FUNCTION_BLOCK FB_System_FBT_425
VAR_INPUT
	Betrieb_Anford_auto		: BOOL;
	Regelung_Modus_auto		: USINT;
	Regelung_Sollw_auto		: REAL;
	Temp_Aussen				: REAL;
	Temp_Innen				: REAL;
END_VAR
VAR_OUTPUT
	{attribute 'OPC.UA.DA' := '1'}Steuerung				: ST_System_FBT_Steuerung;		
	{attribute 'OPC.UA.DA' := '1'}Stellwert				: ST_System_FBT_Stellwert;		
	{attribute 'OPC.UA.DA' := '1'}Zustand					: ST_System_FBT_Zustand;	
	{attribute 'OPC.UA.DA' := '1'}Parameter				: ST_System_FBT_Parameter;		
END_VAR
VAR
	Pumpe_425				: FB_PU;
	Stellventil_423			: FB_SVs;
	Stellventil_424			: FB_SVs;
	Regelventil_425			: FB_RV;

	Zustandscheck			: FB_System_FBT_Zustandscheck;
	Logik					: FB_System_FBT_Logik;
	Ablaufsteuerung			: FB_System_FBT_Ablaufsteuerung;
	Sollwertscheck			: FB_System_FBT_Sollwertscheck;
	Regelung				: FB_System_FBT_Regelung;
	Stellwertscheck			: FB_System_FBT_Stellwertscheck;

END_VAR
VAR // added by the converter: edge detectors and wires of the graphical bodies
    _w1, _w2 : ANY;
END_VAR

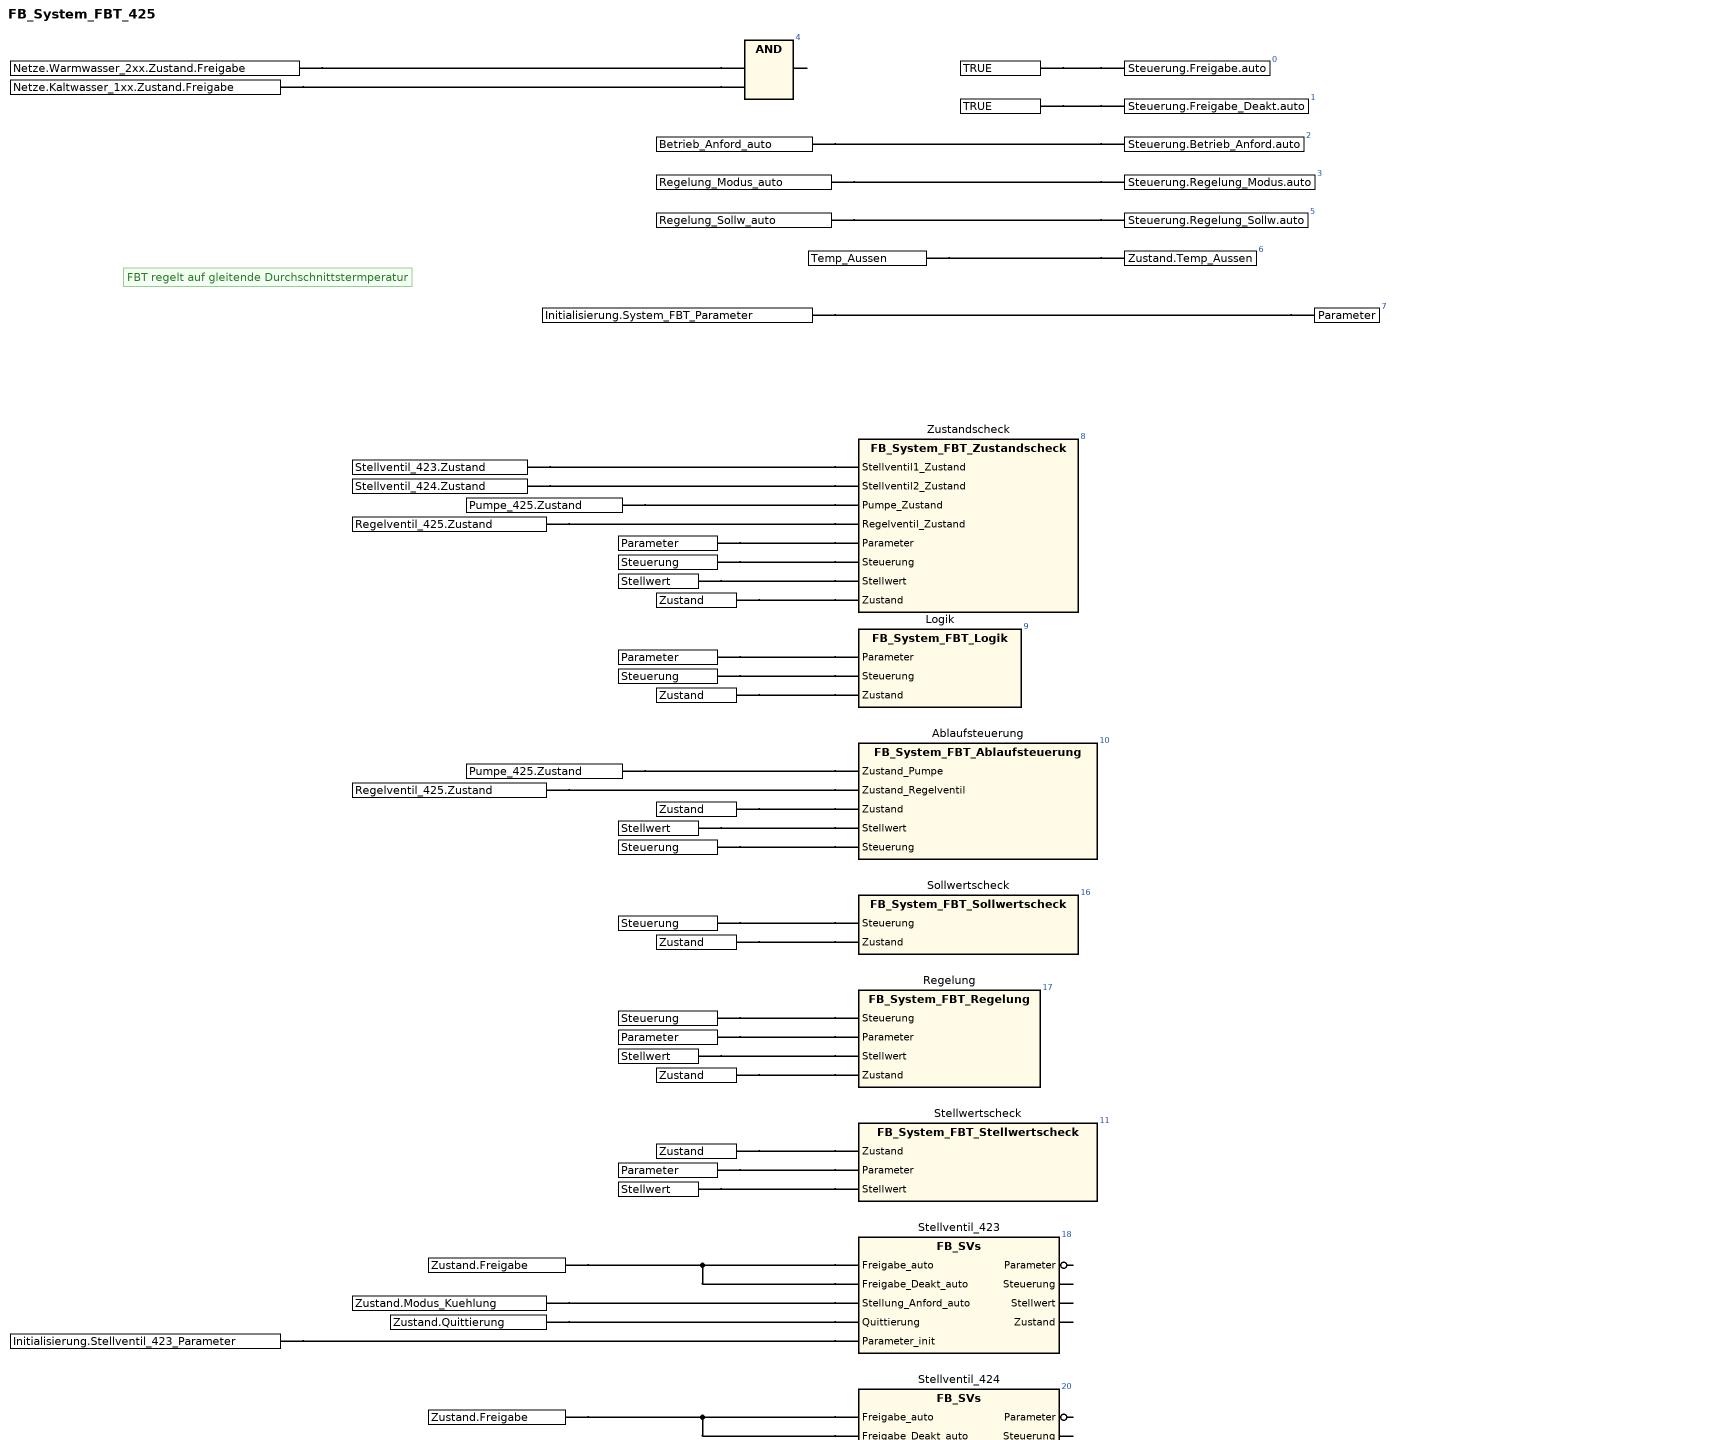
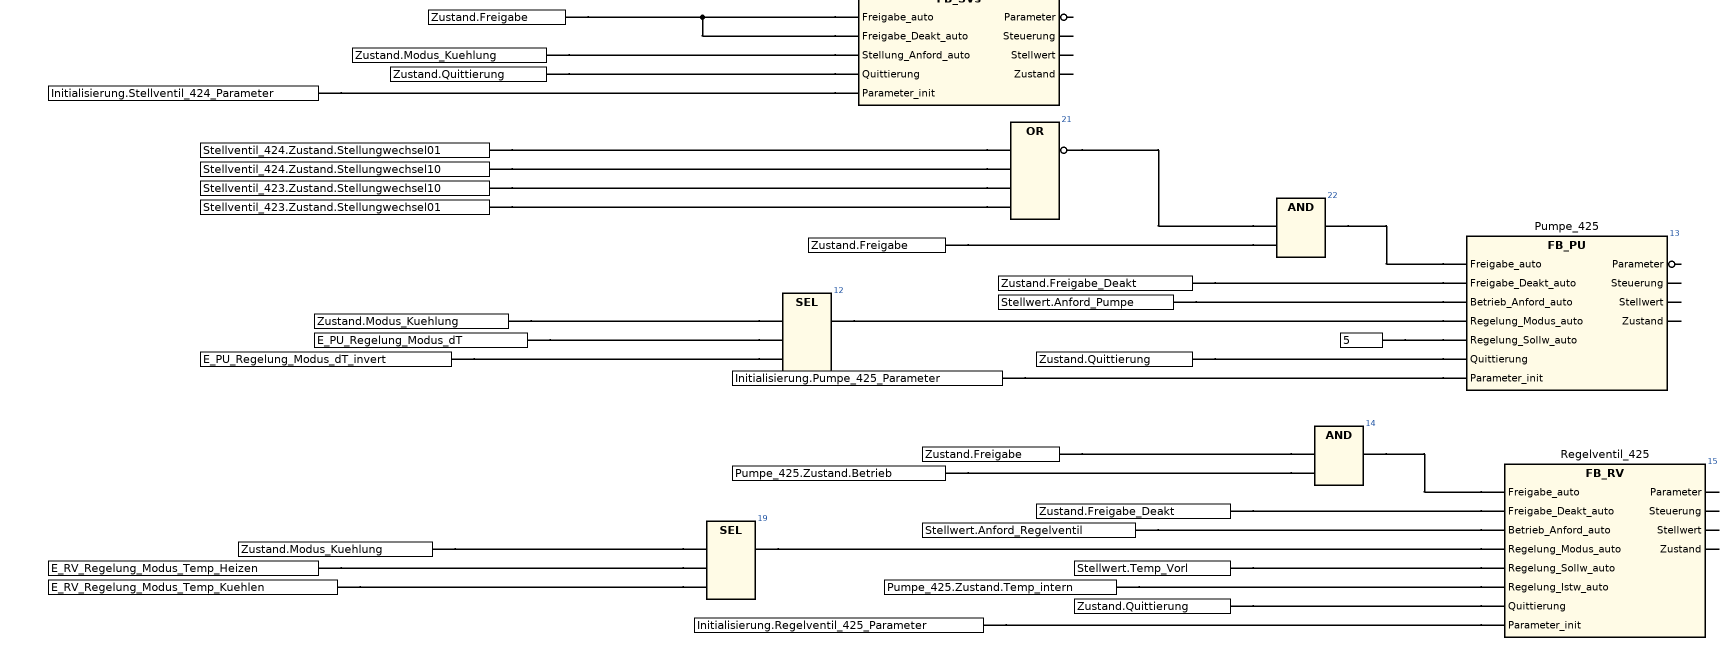
Steuerung.Freigabe.auto := TRUE;
Steuerung.Freigabe_Deakt.auto := TRUE;
Steuerung.Betrieb_Anford.auto := Betrieb_Anford_auto;
Steuerung.Regelung_Modus.auto := Regelung_Modus_auto;
(* Netze.Warmwasser_2xx.Zustand.Freigabe AND Netze.Kaltwasser_1xx.Zustand.Freigabe; result not used *)
Steuerung.Regelung_Sollw.auto := Regelung_Sollw_auto;
Zustand.Temp_Aussen := Temp_Aussen;
Parameter := Initialisierung.System_FBT_Parameter;
// FBT regelt auf gleitende Durchschnittstermperatur
Zustandscheck(
    Stellventil1_Zustand := Stellventil_423.Zustand,
    Stellventil2_Zustand := Stellventil_424.Zustand,
    Pumpe_Zustand := Pumpe_425.Zustand,
    Regelventil_Zustand := Regelventil_425.Zustand,
    Parameter := Parameter,
    Steuerung := Steuerung,
    Stellwert := Stellwert,
    Zustand := Zustand); // FB_System_FBT_Zustandscheck
Logik(Parameter := Parameter, Steuerung := Steuerung, Zustand := Zustand); // FB_System_FBT_Logik
Ablaufsteuerung(
    Zustand_Pumpe := Pumpe_425.Zustand,
    Zustand_Regelventil := Regelventil_425.Zustand,
    Zustand := Zustand,
    Stellwert := Stellwert,
    Steuerung := Steuerung); // FB_System_FBT_Ablaufsteuerung
Stellwertscheck(Zustand := Zustand, Parameter := Parameter, Stellwert := Stellwert); // FB_System_FBT_Stellwertscheck
Pumpe_425(
    Freigabe_auto := _w1,
    Freigabe_Deakt_auto := Zustand.Freigabe_Deakt,
    Betrieb_Anford_auto := Stellwert.Anford_Pumpe,
    Regelung_Modus_auto := SEL(Zustand.Modus_Kuehlung, E_PU_Regelung_Modus_dT, E_PU_Regelung_Modus_dT_invert),
    Regelung_Sollw_auto := 5,
    Quittierung := Zustand.Quittierung,
    Parameter_init := Initialisierung.Pumpe_425_Parameter); // FB_PU
Regelventil_425(
    Freigabe_auto := Zustand.Freigabe AND Pumpe_425.Zustand.Betrieb,
    Freigabe_Deakt_auto := Zustand.Freigabe_Deakt,
    Betrieb_Anford_auto := Stellwert.Anford_Regelventil,
    Regelung_Modus_auto := _w2,
    Regelung_Sollw_auto := Stellwert.Temp_Vorl,
    Regelung_Istw_auto := Pumpe_425.Zustand.Temp_intern,
    Quittierung := Zustand.Quittierung,
    Parameter_init := Initialisierung.Regelventil_425_Parameter); // FB_RV
Sollwertscheck(Steuerung := Steuerung, Zustand := Zustand); // FB_System_FBT_Sollwertscheck
Regelung(Steuerung := Steuerung, Parameter := Parameter, Stellwert := Stellwert, Zustand := Zustand); // FB_System_FBT_Regelung
Stellventil_423(
    Freigabe_auto := Zustand.Freigabe,
    Freigabe_Deakt_auto := Zustand.Freigabe,
    Stellung_Anford_auto := Zustand.Modus_Kuehlung,
    Quittierung := Zustand.Quittierung,
    Parameter_init := Initialisierung.Stellventil_423_Parameter); // FB_SVs
_w2 := SEL(Zustand.Modus_Kuehlung, E_RV_Regelung_Modus_Temp_Heizen, E_RV_Regelung_Modus_Temp_Kuehlen);
Stellventil_424(
    Freigabe_auto := Zustand.Freigabe,
    Freigabe_Deakt_auto := Zustand.Freigabe,
    Stellung_Anford_auto := Zustand.Modus_Kuehlung,
    Quittierung := Zustand.Quittierung,
    Parameter_init := Initialisierung.Stellventil_424_Parameter); // FB_SVs
_w1 := NOT (Stellventil_424.Zustand.Stellungwechsel01 OR Stellventil_424.Zustand.Stellungwechsel10 OR Stellventil_423.Zustand.Stellungwechsel10 OR Stellventil_423.Zustand.Stellungwechsel01) AND Zustand.Freigabe;

END_FUNCTION_BLOCK

(* stored: Version 1.1.0.1, ProductVersion 3.1.4024.9
   POU FB_System_FBT_425: Id {4ad62e70-8f83-46e7-91e5-240c94957bd5}, SpecialFunc None *)
